Staubli VAL3: getItem.pgx

public program getItem(InstrItem& x_sItem (dimensions=1), num x_nIndex (dimensions=1))
begin
  // give back the instruction
  x_sItem=pEdit.iEvent[x_nIndex]
end
